TYPE ST_ReadSingleOffsetData_Status EXTENDS ST_StatusBasic :
STRUCT
END_STRUCT
END_TYPE

(* stored: Version 1.1.0.1, ProductVersion 3.1.4024.13
   DUT ST_ReadSingleOffsetData_Status: Id {6cc0c3ce-6356-4731-b390-84c6c6f55ca5} *)
